FUNCTION_BLOCK _LREAL_TestSuite EXTENDS TcUnit.FB_TestSuite
VAR
END_VAR

TestAddress();
TestClearReference();
TestClone();
TestTypeNameReturnsExpected();
TestIsFloat();
TestIsSigned();
TestMakeReferenceToFollowsReference();
TestMakeReferenceToUpdatesReference();
TestSize();
TestValueReturnsExpectedAfterInit();
TestValueReturnsExpectedAfterChange();
TestSerializeTypeWith();
TestSerializeWith();
TestTryDeserializeFrom();
TestTryMakeReferenceToFollowsReference();
TestTryMakeReferenceToUpdatesReference();

METHOD PUBLIC TestAddress
VAR
    _type : _LREAL(0.0);
    notExpected : PVOID := 0;
    actual : PVOID;
END_VAR
TEST('TestAddress');

actual := _type.Address;

AssertFalse(
    Condition := (notExpected = actual),
    Message := 'Type did not return a valid address.'
);

TEST_FINISHED();
END_METHOD

METHOD PUBLIC TestClearReference
VAR
    _type : _LREAL(0.0);
	target : LREAL := 0.0;
    expected : LREAL := 0.0;
    actual : LREAL;
END_VAR
TEST('TestClearReference');

_type.MakeReferenceTo(target);
_type.ClearReference();
target := 123.4;

actual := _type.Value;

AssertEquals_LREAL(
    Expected := expected,
    Actual := actual,
    Delta := LREAL#0.001,
    Message := 'Value did not follow target change'
);

TEST_FINISHED();
END_METHOD

METHOD PUBLIC TestClone
VAR
    _type : _LREAL(123.4);
	clone : I_Datatype;
	isValidClone : BOOL;
	compareResult : DINT;
END_VAR
TEST('TestClone');

clone := _type.Clone();

isValidClone := clone <> 0;

IF isValidClone THEN
	compareResult := memcmp(_type.Address, clone.Address, clone.Size);
END_IF

AssertTrue(
	Condition := isValidClone,
	Message := 'Clone did not produce a clone'
);

AssertEquals_DINT(
	Expected := 0,
    Actual := compareResult,
    Message := 'Clone did not return a valid clone.'
);

clone.Dispose();

TEST_FINISHED();
END_METHOD

METHOD PUBLIC TestIsFloat
VAR
    _type : _LREAL(0);
END_VAR
TEST('TestIsFloat');

AssertTrue(
	Condition := _type.IsFloat,
    Message := 'Type did not correctly identify itself as being unsigned'
);

TEST_FINISHED();
END_METHOD

METHOD PUBLIC TestIsSigned
VAR
    _type : _LREAL(0);
END_VAR
TEST('TestIsSigned');

AssertTrue(
	Condition := _type.IsSigned,
    Message := 'Type did not correctly identify itself as being signed'
);

TEST_FINISHED();
END_METHOD

METHOD PUBLIC TestMakeReferenceToFollowsReference
VAR
    _type : _LREAL(0.0);
	target : LREAL := 0.0;
    expected : LREAL := 123.4;
    actual : LREAL;
END_VAR
TEST('TestMakeReferenceToFollowsReference');

_type.MakeReferenceTo(target);
target := 123.4;

actual := _type.Value;

AssertEquals_LREAL(
    Expected := expected,
    Actual := actual,
    Delta := LREAL#0.001,
    Message := 'Value did not follow target change'
);

TEST_FINISHED();
END_METHOD

METHOD PUBLIC TestMakeReferenceToUpdatesReference
VAR
    _type : _LREAL(0.0);
	target : LREAL := 0.0;
    expected : LREAL := 123.4;
    actual : LREAL;
END_VAR
TEST('TestMakeReferenceToUpdatesReference');

_type.MakeReferenceTo(target);
_type.Value := 123.4;

actual := target;

AssertEquals_LREAL(
    Expected := expected,
    Actual := actual,
    Delta := LREAL#0.001,
    Message := 'Value did not update target'
);

TEST_FINISHED();
END_METHOD

METHOD PUBLIC TestSerializeTypeWith
VAR
    _type : _LREAL(0.0);
    serializer : JsonSerializer;
    expected : STRING(500) := '{"typeName":"LREAL","minValue":-1.7976931348623157e308,"maxValue":1.7976931348623157e308,"isSigned":true,"isFloat":true}';
    actual : STRING(500);
END_VAR
TEST('TestSerializeTypeWith');

serializer.Reset();
_type.SerializeTypeWith(serializer);
serializer.TryGetSerializedData(ADR(actual), SIZEOF(actual));

AssertEquals_STRING(
    Expected := expected,
    Actual := actual,
    Message := 'Serialization of type did not return correct string.'
);

TEST_FINISHED();
END_METHOD

METHOD PUBLIC TestSerializeWith
VAR
    _type : _LREAL(123.4);
    serializer : JsonSerializer;
    expected : STRING := '123.4';
    actual : STRING(500);
END_VAR
TEST('TestSerializeWith');

serializer.Reset();
_type.SerializeWith(serializer);
serializer.TryGetSerializedData(ADR(actual), SIZEOF(actual));

AssertEquals_STRING(
    Expected := expected,
    Actual := actual,
    Message := 'Serialization of type data did not return correct string.'
);

TEST_FINISHED();
END_METHOD

METHOD PUBLIC TestSize
VAR
    _type : _LREAL(0.0);
    expected : UDINT := SIZEOF(LREAL);
    actual : UDINT;
END_VAR
TEST('TestSize');

actual := _type.Size;

AssertEquals_UDINT(
    Expected := Expected,
    Actual := actual,
    Message := 'Type did not return the correct size.'
);

TEST_FINISHED();
END_METHOD

METHOD PUBLIC TestTryDeserializeFrom
VAR
    deserializer : JsonDeserializer;
    feedback : DeserializerFeedback;
    json : STRING := '123.4';
    _type : _LREAL(0.0);
    expected : LREAL := 123.4;
    actual : LREAL;
 END_VAR
TEST('TestTryDeserializeFrom');

deserializer.Reset();
deserializer.TryLoad(json);
_type.TryDeserializeFrom(Deserializer, Feedback);

actual := _type.Value;

AssertEquals_LREAL(
    Expected := expected,
    Actual := actual,
    Delta := LREAL#0.001,
    Message := 'Type did not deserialize correctly.'
);

TEST_FINISHED();
END_METHOD

METHOD PUBLIC TestTryMakeReferenceToFollowsReference
VAR
    _type : _LREAL(0.0);
	target : _LREAL(0.0);
    expected : LREAL := 123.4;
    actual : LREAL;
END_VAR
TEST('TestTryMakeReferenceToFollowsReference');

_type.TryMakeReferenceTo(target);
target.Value := 123.4;

actual := _type.Value;

AssertEquals_LREAL(
    Expected := expected,
    Actual := actual,
    Delta := LREAL#0.001,
    Message := 'Value did not follow target change'
);

TEST_FINISHED();
END_METHOD

METHOD PUBLIC TestTryMakeReferenceToUpdatesReference
VAR
    _type : _LREAL(0.0);
	target : _LREAL(0.0);
    expected : LREAL := 123.4;
    actual : LREAL;
END_VAR
TEST('TestTryMakeReferenceToUpdatesReference');

_type.TryMakeReferenceTo(target);
_type.Value := 123.4;

actual := target.Value;

AssertEquals_LREAL(
    Expected := expected,
    Actual := actual,
    Delta := LREAL#0.001,
    Message := 'Value did not update target'
);

TEST_FINISHED();
END_METHOD

METHOD PUBLIC TestTypeNameReturnsExpected
VAR
    _type : _LREAL(0.0);
    expected : STRING := 'LREAL';
    actual : STRING;
END_VAR
TEST('TestTypeNameReturnsExpected');

actual := _type.TypeName;

AssertEquals_STRING(
    Expected := expected,
    Actual := actual,
    Message := 'Type did not return correct iec type.'
);

TEST_FINISHED();
END_METHOD

METHOD PUBLIC TestValueReturnsExpectedAfterChange
VAR
    _type : _LREAL(0.0);
    expected : LREAL := 123.4;
    actual : LREAL;
END_VAR
TEST('TestValueReturnsExpectedAfterChange');

_type.Value := 123.4;

actual := _type.Value;

AssertEquals_LREAL(
    Expected := expected,
    Actual := actual,
    Delta := LREAL#0.001,
    Message := 'Expected value not returned after change.'
);

TEST_FINISHED();
END_METHOD

METHOD PUBLIC TestValueReturnsExpectedAfterInit
VAR
    _type : _LREAL(123.4);
    expected : LREAL := 123.4;
    actual : LREAL;
END_VAR
TEST('TestValueReturnsExpectedAfterInit');

actual := _type.Value;

AssertEquals_LREAL(
    Expected := expected,
    Actual := actual,
    Delta := LREAL#0.001,
    Message := 'Expected value not returned after Init.'
);

TEST_FINISHED();
END_METHOD

END_FUNCTION_BLOCK

(* stored: Version 1.1.0.1, ProductVersion 3.1.4024.12
   POU _LREAL_TestSuite: Id {226b9966-175f-4f83-8f37-d2ec8549de8b}, SpecialFunc None
   Method TestAddress: Id {0deca302-9b6a-4de2-ab70-33f6c9203c4d}
   Method TestClearReference: Id {fd977c27-7a28-42ae-a15d-1f4e1f19a201}
   Method TestClone: Id {656d1b83-5a6f-4888-b63c-b0e1e9defa27}
   Method TestIsFloat: Id {2978f98f-d661-0bac-398e-04e44cfc0d58}
   Method TestIsSigned: Id {e76cab8e-cac5-432f-bcd0-cfd4c922f4cf}
   Method TestMakeReferenceToFollowsReference: Id {7c4156e6-691c-40f7-b5eb-0b4143a4cb27}
   Method TestMakeReferenceToUpdatesReference: Id {a6764ec9-22a9-4416-9683-5d5e924bafff}
   Method TestSerializeTypeWith: Id {cb749b6f-62b5-4317-8cb3-9109c7960efc}
   Method TestSerializeWith: Id {491bee2c-6380-4b5f-b895-4bf5d6ea940b}
   Method TestSize: Id {3a7198f9-a6a7-4e6b-9ba0-35dfbf53322d}
   Method TestTryDeserializeFrom: Id {3d1b0211-6133-4806-9854-23f8d5e66059}
   Method TestTryMakeReferenceToFollowsReference: Id {b2ff03f7-2a39-4840-9e8f-0a83c7556887}
   Method TestTryMakeReferenceToUpdatesReference: Id {c8cc83a6-49de-442c-90ec-c7ef4f28809c}
   Method TestTypeNameReturnsExpected: Id {bb62feec-8447-417a-aaa3-26085a8229c9}
   Method TestValueReturnsExpectedAfterChange: Id {7bba9e58-17dc-4370-8e99-1812866319d2}
   Method TestValueReturnsExpectedAfterInit: Id {bc4dd4e2-1155-4d4f-aa39-f283b249e6f5} *)
